{attribute 'pack_mode' := '1'}
TYPE TMachineManual :
STRUCT
	bCanLockDoor		: BOOL;
	bLockDoor			: BOOL;
	bCanUnlockDoor		: BOOL;
	bUnlockDoor			: BOOL;
END_STRUCT
END_TYPE

(* stored: Version 1.1.0.1, ProductVersion 3.1.4022.12
   DUT TMachineManual: Id {a419da96-579c-4031-a762-f15ca15f1bc1} *)
